Staubli VAL3: goTo.pgx

program goTo(num x_nIndex, bool& x_bUnreached[])
  local bool l_bUnreached
  local num l_nIndexTool
  local tool l_tTool
  local num l_nMoveType
  local mdesc l_mDesc
begin
//  // look for not cycle mode
//  if !cycleStatus:bCycle
//    if cycleStatus:nWorkingMode==1 and isPowered()
//      // check for the index
//      if nOldIndex!=x_nIndex or (cycleStatus:nWorkingStatus!=0 and cycleStatus:nWorkingStatus!=6)
//        if !isEmpty()
//          resetMotion()
//        endIf
//        if nOldIndex!=x_nIndex
//          nOldIndex=x_nIndex
//        endIf
//      else
//        if isEmpty() and cycleStatus:nWorkingStatus==0
//          // get the data to move
//          call trajType:getTool(l_nIndexTool)
//          call tcp:getTool(l_tTool,l_nIndexTool)
//          call trajType:getTrajItem(l_tTraj,x_nIndex)
//          //
//          // use a sTemp mdesc to set the blend off
//          //
//          l_tTraj.nom_speed.blend=off
//          call trajType:goTo(l_tTool,l_tTraj.nom_speed,l_tTraj.moveType,x_bUnreached,x_nIndex)
//          call showPoint()
//        endIf
//      endIf
//    else
//      if cycleStatus:nWorkingMode!=1
//        resetMotion()
//      endIf
//    endIf
//  endIf
end
